// TIA Portal V19 program export: 1 tag tables, 0 data types, 0 data blocks, 3 code blocks (in call order from the OBs), 14 instance data blocks

VAR_GLOBAL   // PLC tag table "Default tag table"
   Axis_1_Drive_IN AT %I68.0 : "PD_TEL3_IN";
   Axis_1_Drive_OUT AT %Q82.0 : "PD_TEL3_OUT";
   "Axis_1_Homing switch" AT %I0.3 : Bool;
   firstscan AT %M10.0 : Bool;
   "Homing procedure" AT %M11.0 : Bool;
   Home_Done_Vertical AT %M11.1 : Bool;
   Tag_1 AT %I2.0 : Bool;
   Tag_2 AT %M20.0 : Bool;
   ServoONHorizont AT %Q0.7 : Bool;
   home_horizontal AT %Q0.4 : Bool;
   Home_done_horizontal AT %M12.0 : Bool;
   HomeComplete AT %I8.0 : Bool;
   Tag_3 AT %I1.3 : Bool;
   Servo_fault AT %I1.4 : Bool;
   Servo_Alarm AT %I1.5 : Bool;
   Tag_4 AT %M100.0 : Bool;
   System_Byte AT %MB8001 : Byte;
   "FirstScan(1)" AT %M1.0 : Bool;
   DiagStatusUpdate AT %M8001.1 : Bool;
   AlwaysTRUE AT %M8001.2 : Bool;
   AlwaysFALSE AT %M8001.3 : Bool;
   Clock_Byte AT %MB8000 : Byte;
   Clock_10Hz AT %M8000.0 : Bool;
   Clock_5Hz AT %M8000.1 : Bool;
   "Clock_2.5Hz" AT %M8000.2 : Bool;
   Clock_2Hz AT %M8000.3 : Bool;
   "Clock_1.25Hz" AT %M8000.4 : Bool;
   Clock_1Hz AT %M8000.5 : Bool;
   "Clock_0.625Hz" AT %M8000.6 : Bool;
   "Clock_0.5Hz" AT %M8000.7 : Bool;
   Tag_5 AT %M100.1 : Bool;
   Reset_HorizontDrive AT %Q0.6 : Bool;
   "hent 8cm" AT %M1000.0 : Bool;
   Binær_hent_8cm AT %M50.0 : Bool;
   Stepdata_1_U AT %Q0.1 : Bool;
   Stepdata_2_U AT %Q0.2 : Bool;
   Stepdata_3_U AT %Q0.3 : Bool;
   Stepdata_1_Conf AT %I0.6 : Bool;
   Stepdata_2_Conf AT %I0.7 : Bool;
   Stepdata_3_Conf AT %I1.0 : Bool;
   Drive_Servo AT %Q0.5 : Bool;
   lever_8cm AT %M1000.1 : Bool;
   "binær _lever_8cm" AT %M50.1 : Bool;
   "Sett sylinder C7" AT %M50.7 : Bool;
   "Sylinder C7" AT %Q0.0 : Bool;
   Tag_8 AT %M50.2 : Bool;
   Hent_16cm AT %M50.4 : Bool;
   Binær_Hent_16cm AT %M50.5 : Bool;
   Lever_16cm AT %M50.6 : Bool;
   binær_lever_16cm AT %M51.0 : Bool;
END_VAR

ORGANIZATION_BLOCK "Main"   // OB1, LAD, ProgramCycle
TITLE = "Main Program Sweep (Cycle)"
{ S7_Optimized_Access := 'TRUE' }
// stored: SetENOAutomatically false
   VAR_INPUT
      Initial_Call : Bool;   // Initial call of this OB
      Remanence : Bool;   // =True, if remanent data are available
   END_VAR
   VAR_TEMP   // added for the SCL form of the ladder/FBD networks
      _w1 : Bool;
   END_VAR
BEGIN

REGION Network 1: Homing Vertical
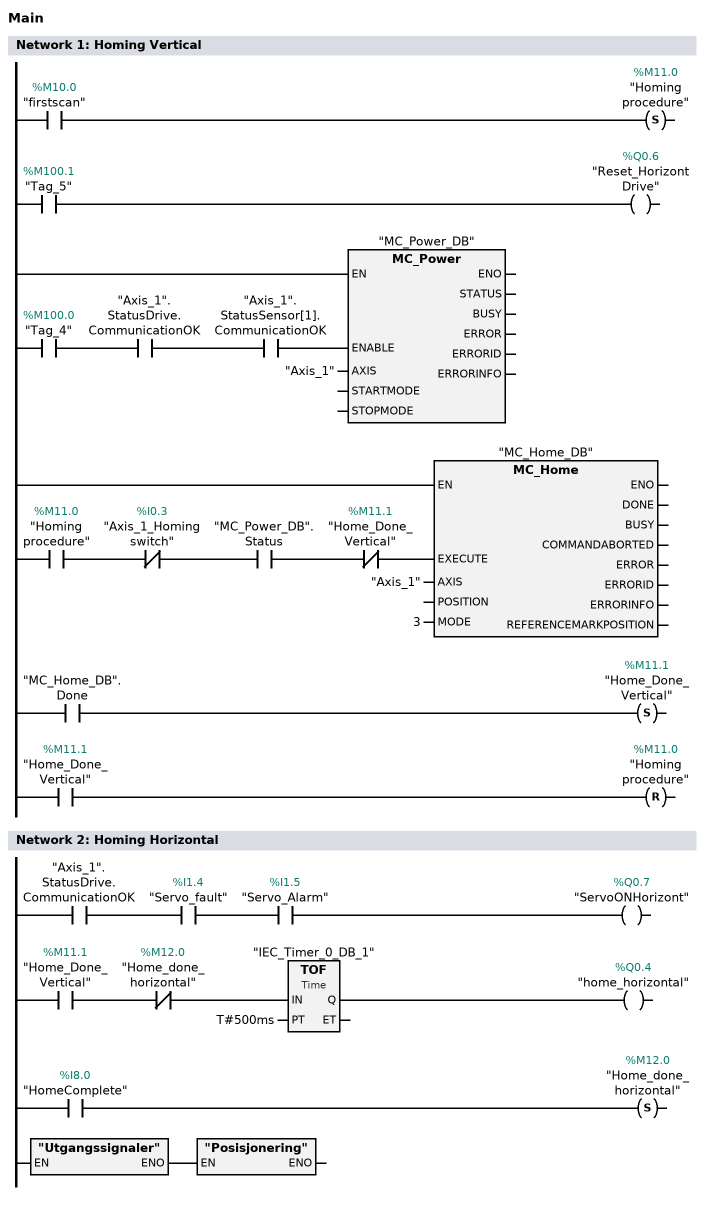
   RUNG wire#powerrail
      Contact( "firstscan" )
      S_Coil( "Homing procedure" )
   END_RUNG
   RUNG wire#powerrail
      Contact( "Tag_5" )
      Coil( "Reset_HorizontDrive" )
   END_RUNG
   RUNG wire#powerrail
      "MC_Power_DB".MC_Power(Enable := wire#w1, Axis := "Axis_1", StartMode :=, StopMode :=, Status =>, Busy =>, Error =>, ErrorID =>, ErrorInfo =>)
   END_RUNG
   RUNG wire#powerrail
      Contact( "Tag_4" )
      Contact( "Axis_1".StatusDrive.CommunicationOK )
      Contact( "Axis_1".StatusSensor[1].CommunicationOK )
   END_RUNG wire#w1
   RUNG wire#powerrail
      "MC_Home_DB".MC_Home(Execute := wire#w2, Axis := "Axis_1", Position :=, Mode := 3, Done =>, Busy =>, CommandAborted =>, Error =>, ErrorID =>, ErrorInfo =>, ReferenceMarkPosition =>)
   END_RUNG
   RUNG wire#powerrail
      Contact( "Homing procedure" )
      I_Contact( "Axis_1_Homing switch" )
      Contact( "MC_Power_DB".Status )
      I_Contact( "Home_Done_Vertical" )
   END_RUNG wire#w2
   RUNG wire#powerrail
      Contact( "MC_Home_DB".Done )
      S_Coil( "Home_Done_Vertical" )
   END_RUNG
   RUNG wire#powerrail
      Contact( "Home_Done_Vertical" )
      R_Coil( "Homing procedure" )
   END_RUNG
   // the same network as SCL:
   IF "firstscan" THEN "Homing procedure" := TRUE; END_IF;
   "Reset_HorizontDrive" := "Tag_5";
   "MC_Power_DB"(Enable := "Tag_4" AND "Axis_1".StatusDrive.CommunicationOK AND "Axis_1".StatusSensor[1].CommunicationOK,   // MC_Power
                 Axis := "Axis_1");
   "MC_Home_DB"(Execute := "Homing procedure" AND NOT "Axis_1_Homing switch" AND "MC_Power_DB".Status AND NOT "Home_Done_Vertical",   // MC_Home
                Axis := "Axis_1",
                Mode := 3);
   IF "MC_Home_DB".Done THEN "Home_Done_Vertical" := TRUE; END_IF;
   IF "Home_Done_Vertical" THEN "Homing procedure" := FALSE; END_IF;
END_REGION

REGION Network 2: Homing Horizontal
   RUNG wire#powerrail
      Contact( "Axis_1".StatusDrive.CommunicationOK )
      Contact( "Servo_fault" )
      Contact( "Servo_Alarm" )
      Coil( "ServoONHorizont" )
   END_RUNG
   RUNG wire#powerrail
      Contact( "Home_Done_Vertical" )
      I_Contact( "Home_done_horizontal" )
      { S7_Templates := "time_type := Time" } "IEC_Timer_0_DB_1".TOF(pt := T#500ms, et =>)
      Coil( "home_horizontal" )
   END_RUNG
   RUNG wire#powerrail
      Contact( "HomeComplete" )
      S_Coil( "Home_done_horizontal" )
   END_RUNG
   RUNG wire#powerrail
      "Utgangssignaler"()
      "Posisjonering"()
   END_RUNG
   // the same network as SCL:
   "ServoONHorizont" := "Axis_1".StatusDrive.CommunicationOK AND "Servo_fault" AND "Servo_Alarm";
   "IEC_Timer_0_DB_1".TOF(IN := "Home_Done_Vertical" AND NOT "Home_done_horizontal", PT := T#500ms);
   "home_horizontal" := "IEC_Timer_0_DB_1".Q;
   IF "HomeComplete" THEN "Home_done_horizontal" := TRUE; END_IF;
   "Utgangssignaler"(ENO => #_w1);
   IF #_w1 THEN "Posisjonering"(); END_IF;
END_REGION
END_ORGANIZATION_BLOCK

FUNCTION "Utgangssignaler" : Void   // FC1, LAD
{ S7_Optimized_Access := 'TRUE' }
// stored: SetENOAutomatically false
BEGIN

REGION Network 1
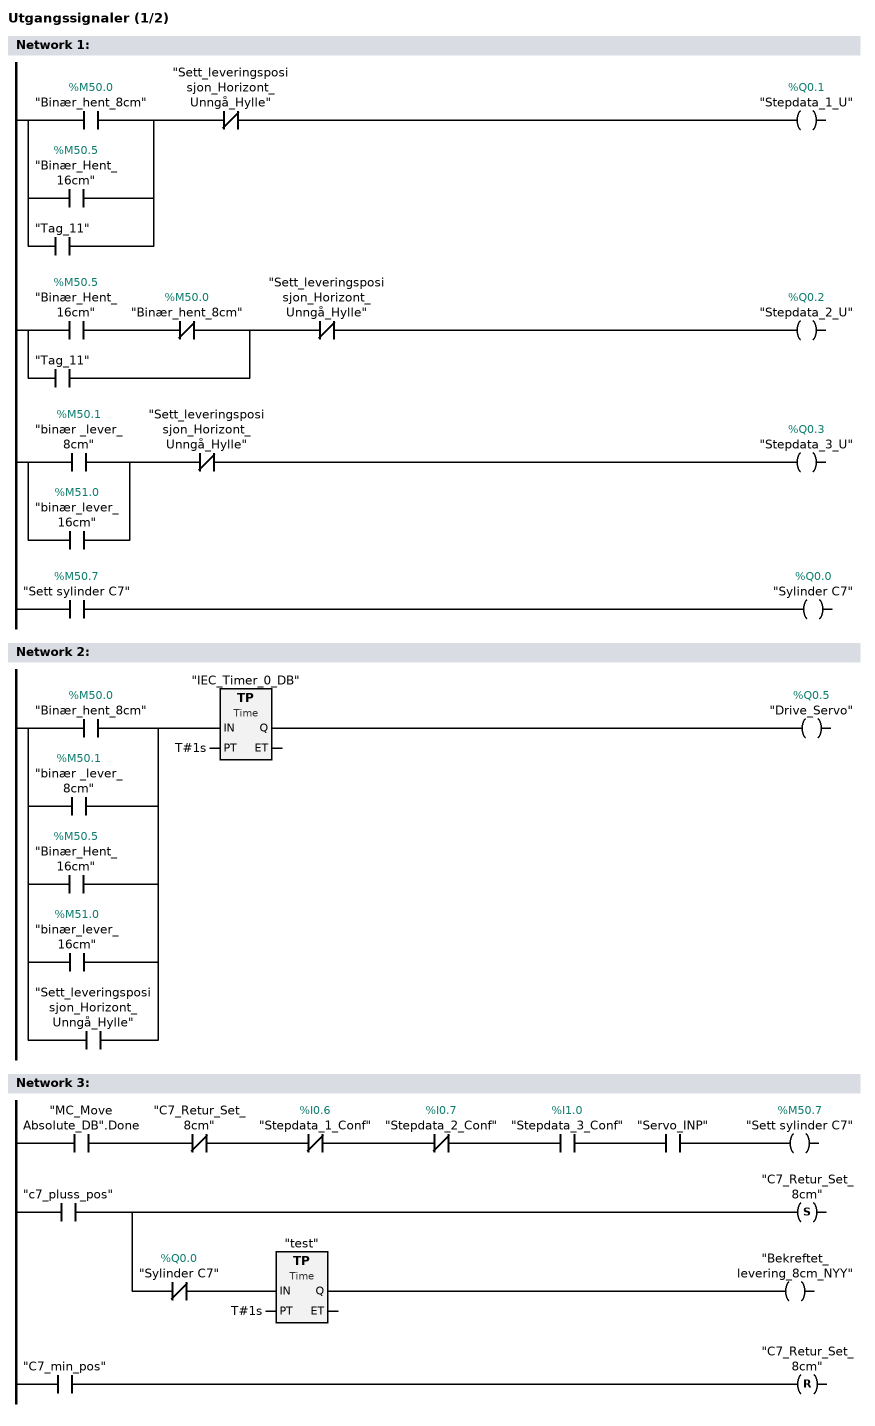
   RUNG wire#powerrail
      Contact( "Binær_hent_8cm" )
      wire#w1
      I_Contact( "Sett_leveringsposisjon_Horizont_Unngå_Hylle" )
      Coil( "Stepdata_1_U" )
   END_RUNG
   RUNG wire#powerrail
      Contact( "Binær_Hent_16cm" )
   END_RUNG wire#w1
   RUNG wire#powerrail
      Contact( "Tag_11" )
   END_RUNG wire#w1
   RUNG wire#powerrail
      Contact( "Binær_Hent_16cm" )
      I_Contact( "Binær_hent_8cm" )
      wire#w2
      I_Contact( "Sett_leveringsposisjon_Horizont_Unngå_Hylle" )
      Coil( "Stepdata_2_U" )
   END_RUNG
   RUNG wire#powerrail
      Contact( "Tag_11" )
   END_RUNG wire#w2
   RUNG wire#powerrail
      Contact( "binær _lever_8cm" )
      wire#w3
      I_Contact( "Sett_leveringsposisjon_Horizont_Unngå_Hylle" )
      Coil( "Stepdata_3_U" )
   END_RUNG
   RUNG wire#powerrail
      Contact( "binær_lever_16cm" )
   END_RUNG wire#w3
   RUNG wire#powerrail
      Contact( "Sett sylinder C7" )
      Coil( "Sylinder C7" )
   END_RUNG
   // the same network as SCL:
   "Stepdata_1_U" := ("Binær_hent_8cm" OR "Binær_Hent_16cm" OR "Tag_11") AND NOT "Sett_leveringsposisjon_Horizont_Unngå_Hylle";
   "Stepdata_2_U" := (("Binær_Hent_16cm" AND NOT "Binær_hent_8cm") OR "Tag_11") AND NOT "Sett_leveringsposisjon_Horizont_Unngå_Hylle";
   "Stepdata_3_U" := ("binær _lever_8cm" OR "binær_lever_16cm") AND NOT "Sett_leveringsposisjon_Horizont_Unngå_Hylle";
   "Sylinder C7" := "Sett sylinder C7";
END_REGION

REGION Network 2
   RUNG wire#powerrail
      Contact( "Binær_hent_8cm" )
      wire#w1
      { S7_Templates := "time_type := Time" } "IEC_Timer_0_DB".TP(pt := T#1s, et =>)
      Coil( "Drive_Servo" )
   END_RUNG
   RUNG wire#powerrail
      Contact( "binær _lever_8cm" )
   END_RUNG wire#w1
   RUNG wire#powerrail
      Contact( "Binær_Hent_16cm" )
   END_RUNG wire#w1
   RUNG wire#powerrail
      Contact( "binær_lever_16cm" )
   END_RUNG wire#w1
   RUNG wire#powerrail
      Contact( "Sett_leveringsposisjon_Horizont_Unngå_Hylle" )
   END_RUNG wire#w1
   // the same network as SCL:
   "IEC_Timer_0_DB".TP(IN := "Binær_hent_8cm" OR "binær _lever_8cm" OR "Binær_Hent_16cm" OR "binær_lever_16cm" OR "Sett_leveringsposisjon_Horizont_Unngå_Hylle",
                       PT := T#1s);
   "Drive_Servo" := "IEC_Timer_0_DB".Q;
END_REGION

REGION Network 3
   RUNG wire#powerrail
      Contact( "MC_MoveAbsolute_DB".Done )
      I_Contact( "C7_Retur_Set_8cm" )
      I_Contact( "Stepdata_1_Conf" )
      I_Contact( "Stepdata_2_Conf" )
      Contact( "Stepdata_3_Conf" )
      Contact( "Servo_INP" )
      Coil( "Sett sylinder C7" )
   END_RUNG
   RUNG wire#powerrail
      Contact( "c7_pluss_pos" )
      wire#w1
      S_Coil( "C7_Retur_Set_8cm" )
   END_RUNG
   RUNG wire#w1
      I_Contact( "Sylinder C7" )
      { S7_Templates := "time_type := Time" } "test".TP(pt := T#1s, et =>)
      Coil( "Bekreftet_levering_8cm_NYY" )
   END_RUNG
   RUNG wire#powerrail
      Contact( "C7_min_pos" )
      R_Coil( "C7_Retur_Set_8cm" )
   END_RUNG
   // the same network as SCL:
   "Sett sylinder C7" := "MC_MoveAbsolute_DB".Done AND NOT "C7_Retur_Set_8cm" AND NOT "Stepdata_1_Conf" AND NOT "Stepdata_2_Conf" AND "Stepdata_3_Conf" AND "Servo_INP";
   IF "c7_pluss_pos" THEN "C7_Retur_Set_8cm" := TRUE; END_IF;
   "test".TP(IN := "c7_pluss_pos" AND NOT "Sylinder C7", PT := T#1s);
   "Bekreftet_levering_8cm_NYY" := "test".Q;
   IF "C7_min_pos" THEN "C7_Retur_Set_8cm" := FALSE; END_IF;
END_REGION

REGION Network 4
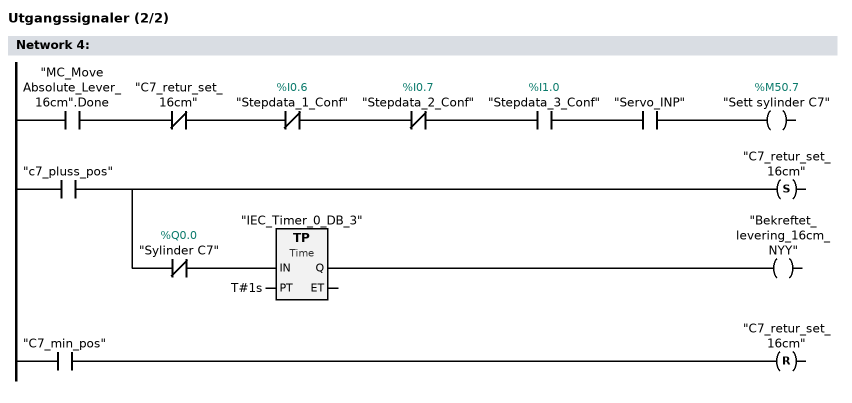
   RUNG wire#powerrail
      Contact( "MC_MoveAbsolute_Lever_16cm".Done )
      I_Contact( "C7_retur_set_16cm" )
      I_Contact( "Stepdata_1_Conf" )
      I_Contact( "Stepdata_2_Conf" )
      Contact( "Stepdata_3_Conf" )
      Contact( "Servo_INP" )
      Coil( "Sett sylinder C7" )
   END_RUNG
   RUNG wire#powerrail
      Contact( "c7_pluss_pos" )
      wire#w1
      S_Coil( "C7_retur_set_16cm" )
   END_RUNG
   RUNG wire#w1
      I_Contact( "Sylinder C7" )
      { S7_Templates := "time_type := Time" } "IEC_Timer_0_DB_3".TP(pt := T#1s, et =>)
      Coil( "Bekreftet_levering_16cm_NYY" )
   END_RUNG
   RUNG wire#powerrail
      Contact( "C7_min_pos" )
      R_Coil( "C7_retur_set_16cm" )
   END_RUNG
   // the same network as SCL:
   "Sett sylinder C7" := "MC_MoveAbsolute_Lever_16cm".Done AND NOT "C7_retur_set_16cm" AND NOT "Stepdata_1_Conf" AND NOT "Stepdata_2_Conf" AND "Stepdata_3_Conf" AND "Servo_INP";
   IF "c7_pluss_pos" THEN "C7_retur_set_16cm" := TRUE; END_IF;
   "IEC_Timer_0_DB_3".TP(IN := "c7_pluss_pos" AND NOT "Sylinder C7", PT := T#1s);
   "Bekreftet_levering_16cm_NYY" := "IEC_Timer_0_DB_3".Q;
   IF "C7_min_pos" THEN "C7_retur_set_16cm" := FALSE; END_IF;
END_REGION
END_FUNCTION

FUNCTION "Posisjonering" : Void   // FC2, LAD
{ S7_Optimized_Access := 'TRUE' }
// stored: SetENOAutomatically false
BEGIN

REGION Network 1
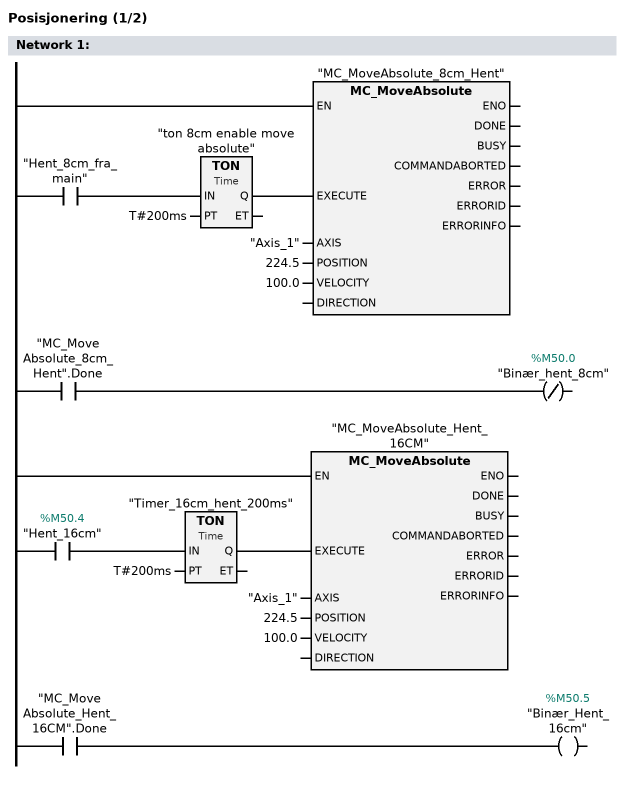
   RUNG wire#powerrail
      "MC_MoveAbsolute_8cm_Hent".MC_MoveAbsolute(Execute := wire#w1, Axis := "Axis_1", Position := 224.5, Velocity := 100.0, Direction :=, Done =>, Busy =>, CommandAborted =>, Error =>, ErrorID =>, ErrorInfo =>)
   END_RUNG
   RUNG wire#powerrail
      Contact( "Hent_8cm_fra_main" )
      { S7_Templates := "time_type := Time" } "ton 8cm enable move absolute".TON(pt := T#200ms, et =>)
   END_RUNG wire#w1
   RUNG wire#powerrail
      Contact( "MC_MoveAbsolute_8cm_Hent".Done )
      I_Coil( "Binær_hent_8cm" )
   END_RUNG
   RUNG wire#powerrail
      "MC_MoveAbsolute_Hent_16CM".MC_MoveAbsolute(Execute := wire#w2, Axis := "Axis_1", Position := 224.5, Velocity := 100.0, Direction :=, Done =>, Busy =>, CommandAborted =>, Error =>, ErrorID =>, ErrorInfo =>)
   END_RUNG
   RUNG wire#powerrail
      Contact( "Hent_16cm" )
      { S7_Templates := "time_type := Time" } "Timer_16cm_hent_200ms".TON(pt := T#200ms, et =>)
   END_RUNG wire#w2
   RUNG wire#powerrail
      Contact( "MC_MoveAbsolute_Hent_16CM".Done )
      Coil( "Binær_Hent_16cm" )
   END_RUNG
   // the same network as SCL:
   "ton 8cm enable move absolute".TON(IN := "Hent_8cm_fra_main", PT := T#200ms);
   "MC_MoveAbsolute_8cm_Hent"(Execute := "ton 8cm enable move absolute".Q,   // MC_MoveAbsolute
                           Axis := "Axis_1",
                           Position := 224.5,
                           Velocity := 100.0);
   "Binær_hent_8cm" := NOT "MC_MoveAbsolute_8cm_Hent".Done;
   "Timer_16cm_hent_200ms".TON(IN := "Hent_16cm", PT := T#200ms);
   "MC_MoveAbsolute_Hent_16CM"(Execute := "Timer_16cm_hent_200ms".Q,   // MC_MoveAbsolute
                           Axis := "Axis_1",
                           Position := 224.5,
                           Velocity := 100.0);
   "Binær_Hent_16cm" := "MC_MoveAbsolute_Hent_16CM".Done;
END_REGION

REGION Network 2
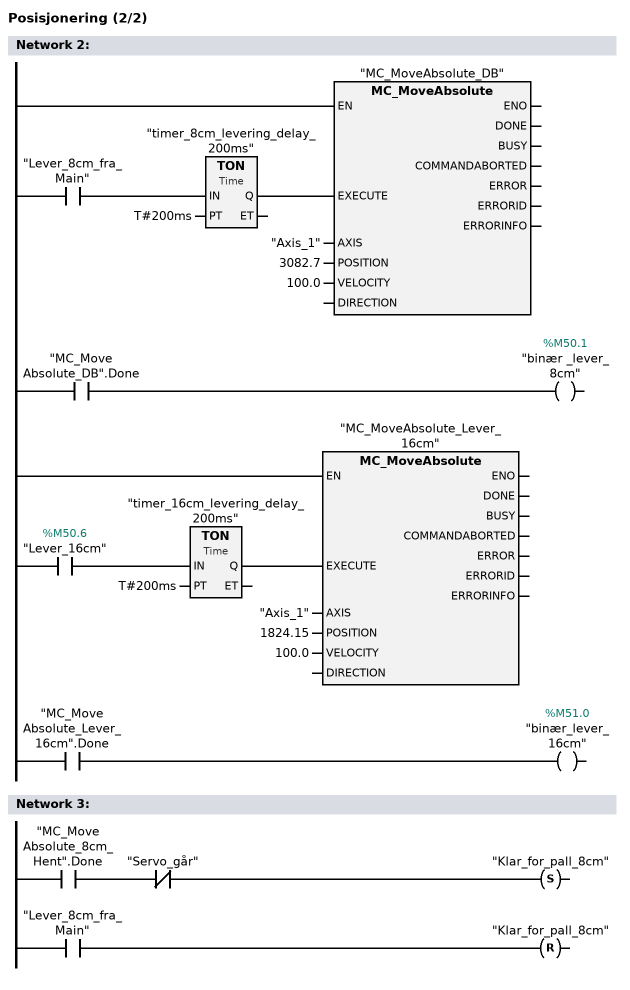
   RUNG wire#powerrail
      "MC_MoveAbsolute_DB".MC_MoveAbsolute(Execute := wire#w1, Axis := "Axis_1", Position := 3082.7, Velocity := 100.0, Direction :=, Done =>, Busy =>, CommandAborted =>, Error =>, ErrorID =>, ErrorInfo =>)
   END_RUNG
   RUNG wire#powerrail
      Contact( "Lever_8cm_fra_Main" )
      { S7_Templates := "time_type := Time" } "timer_8cm_levering_delay_200ms".TON(pt := T#200ms, et =>)
   END_RUNG wire#w1
   RUNG wire#powerrail
      Contact( "MC_MoveAbsolute_DB".Done )
      Coil( "binær _lever_8cm" )
   END_RUNG
   RUNG wire#powerrail
      "MC_MoveAbsolute_Lever_16cm".MC_MoveAbsolute(Execute := wire#w2, Axis := "Axis_1", Position := 1824.15, Velocity := 100.0, Direction :=, Done =>, Busy =>, CommandAborted =>, Error =>, ErrorID =>, ErrorInfo =>)
   END_RUNG
   RUNG wire#powerrail
      Contact( "Lever_16cm" )
      { S7_Templates := "time_type := Time" } "timer_16cm_levering_delay_200ms".TON(pt := T#200ms, et =>)
   END_RUNG wire#w2
   RUNG wire#powerrail
      Contact( "MC_MoveAbsolute_Lever_16cm".Done )
      Coil( "binær_lever_16cm" )
   END_RUNG
   // the same network as SCL:
   "timer_8cm_levering_delay_200ms".TON(IN := "Lever_8cm_fra_Main", PT := T#200ms);
   "MC_MoveAbsolute_DB"(Execute := "timer_8cm_levering_delay_200ms".Q,   // MC_MoveAbsolute
                        Axis := "Axis_1",
                        Position := 3082.7,
                        Velocity := 100.0);
   "binær _lever_8cm" := "MC_MoveAbsolute_DB".Done;
   "timer_16cm_levering_delay_200ms".TON(IN := "Lever_16cm", PT := T#200ms);
   "MC_MoveAbsolute_Lever_16cm"(Execute := "timer_16cm_levering_delay_200ms".Q,   // MC_MoveAbsolute
                           Axis := "Axis_1",
                           Position := 1824.15,
                           Velocity := 100.0);
   "binær_lever_16cm" := "MC_MoveAbsolute_Lever_16cm".Done;
END_REGION

REGION Network 3
   RUNG wire#powerrail
      Contact( "MC_MoveAbsolute_8cm_Hent".Done )
      I_Contact( "Servo_går" )
      S_Coil( "Klar_for_pall_8cm" )
   END_RUNG
   RUNG wire#powerrail
      Contact( "Lever_8cm_fra_Main" )
      R_Coil( "Klar_for_pall_8cm" )
   END_RUNG
   // the same network as SCL:
   IF "MC_MoveAbsolute_8cm_Hent".Done AND NOT "Servo_går" THEN "Klar_for_pall_8cm" := TRUE; END_IF;
   IF "Lever_8cm_fra_Main" THEN "Klar_for_pall_8cm" := FALSE; END_IF;
END_REGION
END_FUNCTION

DATA_BLOCK "Home delay firstscan"   // DB8
{ S7_Optimized_Access := 'TRUE' }
// stored: InstanceOfName IEC_TIMER, OfSystemLibElement IEC_TIMER, OfSystemLibVersion 1.0
"IEC_TIMER"
   // VAR
   //    PT : Time;
   //    ET { ExternalWritable := 'False'} : Time;
   //    IN : Bool;
   //    Q { ExternalWritable := 'False'} : Bool;
   // END_VAR
BEGIN
END_DATA_BLOCK

DATA_BLOCK "IEC_Timer_0_DB"   // DB4
{ S7_Optimized_Access := 'TRUE' }
// stored: InstanceOfName IEC_TIMER, OfSystemLibElement IEC_TIMER, OfSystemLibVersion 1.0
"IEC_TIMER"
   // VAR
   //    PT : Time;
   //    ET { ExternalWritable := 'False'} : Time;
   //    IN : Bool;
   //    Q { ExternalWritable := 'False'} : Bool;
   // END_VAR
BEGIN
END_DATA_BLOCK

DATA_BLOCK "IEC_Timer_0_DB_1"   // DB6
{ S7_Optimized_Access := 'TRUE' }
// stored: InstanceOfName IEC_TIMER, OfSystemLibElement IEC_TIMER, OfSystemLibVersion 1.0
"IEC_TIMER"
   // VAR
   //    PT : Time;
   //    ET { ExternalWritable := 'False'} : Time;
   //    IN : Bool;
   //    Q { ExternalWritable := 'False'} : Bool;
   // END_VAR
BEGIN
END_DATA_BLOCK

DATA_BLOCK "MC_Home_DB"   // DB3
// stored: InstanceOfName MC_Home, OfSystemLibElement MC_Home, OfSystemLibVersion 7.0
"MC_Home"
   // VAR_INPUT
   //    Axis : TO_Axis;
   //    Execute : Bool;
   //    Position : Real;
   //    Mode : Int;
   // END_VAR
   // VAR_OUTPUT
   //    Done : Bool;
   //    Busy : Bool;
   //    CommandAborted : Bool;
   //    Error : Bool;
   //    ErrorID : Word;
   //    ErrorInfo : Word;
   //    ReferenceMarkPosition : Real;
   // END_VAR
   // VAR
   //    FB_ID : DInt;
   // END_VAR
BEGIN
END_DATA_BLOCK

DATA_BLOCK "MC_MoveAbsolute_8cm_Hent"   // DB7
// stored: InstanceOfName MC_MoveAbsolute, OfSystemLibElement MC_MoveAbsolute, OfSystemLibVersion 7.0
"MC_MoveAbsolute"
   // VAR_INPUT
   //    Axis : TO_PositioningAxis;
   //    Execute : Bool;
   //    Position : Real;
   //    Velocity : Real;
   //    Direction : Int;
   // END_VAR
   // VAR_OUTPUT
   //    Done : Bool;
   //    Busy : Bool;
   //    CommandAborted : Bool;
   //    Error : Bool;
   //    ErrorID : Word;
   //    ErrorInfo : Word;
   // END_VAR
   // VAR
   //    FB_ID : DInt;
   // END_VAR
BEGIN
END_DATA_BLOCK

DATA_BLOCK "MC_MoveAbsolute_DB"   // DB9
// stored: InstanceOfName MC_MoveAbsolute, OfSystemLibElement MC_MoveAbsolute, OfSystemLibVersion 7.0
"MC_MoveAbsolute"
   // VAR_INPUT
   //    Axis : TO_PositioningAxis;
   //    Execute : Bool;
   //    Position : Real;
   //    Velocity : Real;
   //    Direction : Int;
   // END_VAR
   // VAR_OUTPUT
   //    Done : Bool;
   //    Busy : Bool;
   //    CommandAborted : Bool;
   //    Error : Bool;
   //    ErrorID : Word;
   //    ErrorInfo : Word;
   // END_VAR
   // VAR
   //    FB_ID : DInt;
   // END_VAR
BEGIN
END_DATA_BLOCK

DATA_BLOCK "MC_MoveAbsolute_Hent_16CM"   // DB11
// stored: InstanceOfName MC_MoveAbsolute, OfSystemLibElement MC_MoveAbsolute, OfSystemLibVersion 7.0
"MC_MoveAbsolute"
   // VAR_INPUT
   //    Axis : TO_PositioningAxis;
   //    Execute : Bool;
   //    Position : Real;
   //    Velocity : Real;
   //    Direction : Int;
   // END_VAR
   // VAR_OUTPUT
   //    Done : Bool;
   //    Busy : Bool;
   //    CommandAborted : Bool;
   //    Error : Bool;
   //    ErrorID : Word;
   //    ErrorInfo : Word;
   // END_VAR
   // VAR
   //    FB_ID : DInt;
   // END_VAR
BEGIN
END_DATA_BLOCK

DATA_BLOCK "MC_MoveAbsolute_Lever_16cm"   // DB13
// stored: InstanceOfName MC_MoveAbsolute, OfSystemLibElement MC_MoveAbsolute, OfSystemLibVersion 7.0
"MC_MoveAbsolute"
   // VAR_INPUT
   //    Axis : TO_PositioningAxis;
   //    Execute : Bool;
   //    Position : Real;
   //    Velocity : Real;
   //    Direction : Int;
   // END_VAR
   // VAR_OUTPUT
   //    Done : Bool;
   //    Busy : Bool;
   //    CommandAborted : Bool;
   //    Error : Bool;
   //    ErrorID : Word;
   //    ErrorInfo : Word;
   // END_VAR
   // VAR
   //    FB_ID : DInt;
   // END_VAR
BEGIN
END_DATA_BLOCK

DATA_BLOCK "MC_Power_DB"   // DB2
// stored: InstanceOfName MC_Power, OfSystemLibElement MC_Power, OfSystemLibVersion 7.0
"MC_Power"
   // VAR_INPUT
   //    Axis : TO_Axis;
   //    Enable : Bool;
   //    StartMode : Int;
   //    StopMode : Int;
   // END_VAR
   // VAR_OUTPUT
   //    Status : Bool;
   //    Busy : Bool;
   //    Error : Bool;
   //    ErrorID : Word;
   //    ErrorInfo : Word;
   // END_VAR
   // VAR
   //    FB_ID : DInt;
   // END_VAR
BEGIN
END_DATA_BLOCK

DATA_BLOCK "Timer_16cm_hent_200ms"   // DB12
{ S7_Optimized_Access := 'TRUE' }
// stored: InstanceOfName IEC_TIMER, OfSystemLibElement IEC_TIMER, OfSystemLibVersion 1.0
"IEC_TIMER"
   // VAR
   //    PT : Time;
   //    ET { ExternalWritable := 'False'} : Time;
   //    IN : Bool;
   //    Q { ExternalWritable := 'False'} : Bool;
   // END_VAR
BEGIN
END_DATA_BLOCK

DATA_BLOCK "timer_16cm_levering_delay_200ms"   // DB14
{ S7_Optimized_Access := 'TRUE' }
// stored: InstanceOfName IEC_TIMER, OfSystemLibElement IEC_TIMER, OfSystemLibVersion 1.0
"IEC_TIMER"
   // VAR
   //    PT : Time;
   //    ET { ExternalWritable := 'False'} : Time;
   //    IN : Bool;
   //    Q { ExternalWritable := 'False'} : Bool;
   // END_VAR
BEGIN
END_DATA_BLOCK

DATA_BLOCK "timer_8cm_levering_delay_200ms"   // DB10
{ S7_Optimized_Access := 'TRUE' }
// stored: InstanceOfName IEC_TIMER, OfSystemLibElement IEC_TIMER, OfSystemLibVersion 1.0
"IEC_TIMER"
   // VAR
   //    PT : Time;
   //    ET { ExternalWritable := 'False'} : Time;
   //    IN : Bool;
   //    Q { ExternalWritable := 'False'} : Bool;
   // END_VAR
BEGIN
END_DATA_BLOCK

DATA_BLOCK "ton 8cm enable move absolute"   // DB5
{ S7_Optimized_Access := 'TRUE' }
// stored: InstanceOfName IEC_TIMER, OfSystemLibElement IEC_TIMER, OfSystemLibVersion 1.0
"IEC_TIMER"
   // VAR
   //    PT : Time;
   //    ET { ExternalWritable := 'False'} : Time;
   //    IN : Bool;
   //    Q { ExternalWritable := 'False'} : Bool;
   // END_VAR
BEGIN
END_DATA_BLOCK

DATA_BLOCK "Axis_1"   // DB1, Motion_DB
AUTHOR : SIMATIC
FAMILY : BasicMC
NAME : TO_PosAx
VERSION : 7.0
// stored: InstanceOfName TO_PositioningAxis, OfSystemLibElement TO_PositioningAxis, OfSystemLibVersion 7.0
TO_PositioningAxis   // technology object, version 7.0
   // // inherited from TO_SpeedAxis
   // // inherited from TO_Axis
   // // inherited from TO_AnyMotionObject
   // VAR
   //    Header : TO_Struct_Header;
   // END_VAR
   // VAR
   //    Position { ExternalWritable := 'False'} : Real;
   //    Velocity { ExternalWritable := 'False'} : Real;
   //    ActualPosition { ExternalWritable := 'False'} : Real;
   //    ActualVelocity { ExternalWritable := 'False'} : Real;
   //    Actor { S7_SetPoint := 'True'} : TO_Struct_Actor;
   //    Sensor { S7_SetPoint := 'True'} : Array[1..1] of TO_Struct_Sensor;
   //    Units { ExternalWritable := 'False'; S7_SetPoint := 'True'} : TO_Struct_Units;
   //    Mechanics { ExternalWritable := 'False'; S7_SetPoint := 'True'} : TO_Struct_Mechanics;
   //    DynamicLimits { ExternalWritable := 'False'; S7_SetPoint := 'True'} : TO_Struct_DynamicLimits;
   //    DynamicDefaults { S7_SetPoint := 'True'} : TO_Struct_DynamicDefaults;
   //    Modulo { ExternalWritable := 'False'; S7_SetPoint := 'True'} : TO_Struct_Modulo;
   //    PositionLimits_SW { S7_SetPoint := 'True'} : TO_Struct_PositionLimitsSW;
   //    PositionLimits_HW { S7_SetPoint := 'True'} : TO_Struct_PositionLimitsHW;
   //    Homing { S7_SetPoint := 'True'} : TO_Struct_Homing;
   //    PositionControl { ExternalWritable := 'False'; S7_SetPoint := 'True'} : TO_Struct_PositionControl;
   //    FollowingError { ExternalWritable := 'False'; S7_SetPoint := 'True'} : TO_Struct_FollowingError;
   //    PositioningMonitoring { ExternalWritable := 'False'; S7_SetPoint := 'True'} : TO_Struct_PositioningMonitoring;
   //    StandstillSignal { ExternalWritable := 'False'; S7_SetPoint := 'True'} : TO_Struct_StandstillSignal;
   //    Simulation { ExternalWritable := 'False'; S7_SetPoint := 'True'} : TO_Struct_Simulation;
   //    StatusPositioning { ExternalWritable := 'False'; S7_SetPoint := 'True'} : TO_Struct_StatusPositioning;
   //    StatusDrive { ExternalWritable := 'False'; S7_SetPoint := 'True'} : TO_Struct_StatusDrive;
   //    StatusSensor { ExternalWritable := 'False'; S7_SetPoint := 'True'} : Array[1..1] of TO_Struct_StatusSensor;
   //    StatusBits { ExternalWritable := 'False'; S7_SetPoint := 'True'} : TO_Struct_StatusBits;
   //    ErrorBits { ExternalWritable := 'False'; S7_SetPoint := 'True'} : TO_Struct_ErrorBits;
   //    ControlPanel { S7_SetPoint := 'True'} : TO_Struct_ControlPanel;
   //    Internal { S7_SetPoint := 'True'} : Array[1..4] of TO_Struct_Internal;
   // END_VAR
BEGIN
   Header.VersionMaj := 7;
   Header.VersionMin := 0;
   Header."Type" := 1;
   Actor."Type" := 1;
   Actor.DataAdaption := 1;
   Actor.Interface.AddressIn.RID := 16#0208_070C;
   Actor.Interface.AddressIn.AREA := 16#81;
   Actor.Interface.AddressIn.OFFSET := 544;
   Actor.Interface.AddressOut.RID := 16#0208_070D;
   Actor.Interface.AddressOut.AREA := 16#82;
   Actor.Interface.AddressOut.OFFSET := 656;
   Actor.DriveParameter.MaxSpeed := 5000.0;
   Sensor[1].DataAdaption := 1;
   Sensor[1].Interface.AddressIn.RID := 16#0208_070C;
   Sensor[1].Interface.AddressIn.AREA := 16#81;
   Sensor[1].Interface.AddressIn.OFFSET := 544;
   Sensor[1].Interface.AddressOut.RID := 16#0208_070D;
   Sensor[1].Interface.AddressOut.AREA := 16#82;
   Sensor[1].Interface.AddressOut.OFFSET := 656;
   Sensor[1].Interface."Type" := 2;
   Sensor[1].Parameter.StepsPerRevolution := 2500;
   Sensor[1].Parameter.FineResolutionXist1 := 2;
   Sensor[1].Parameter.FineResolutionXist2 := 0;
   Sensor[1].Parameter.DeterminableRevolutions := 0;
   Sensor[1].ActiveHoming.DigitalInputAddress.RID := 16#0200_0001;
   Sensor[1].ActiveHoming.DigitalInputAddress.AREA := 16#81;
   Sensor[1].ActiveHoming.DigitalInputAddress.OFFSET := 3;
   Sensor[1].ActiveHoming.SwitchLevel := FALSE;
   DynamicLimits.MinVelocity := 0.0;
   DynamicDefaults.Acceleration := 50.0;
   DynamicDefaults.Deceleration := 50.0;
   DynamicDefaults.EmergencyDeceleration := 125.0;
   Homing.AutoReversal := FALSE;
   Homing.ApproachDirection := FALSE;
   _Sensor[1].ActiveHoming.DigitalInput := Axis_1_Homing switch;
   _Sensor[1].DataAdaptionOffline := True;
   _Sensor[1].Interface.ProfiDriveOutName := Axis_1_Drive_OUT;
   _Sensor[1].Interface.ProfiDriveInName := Axis_1_Drive_IN;
   _Actor.DataAdaptionOffline := True;
   _Actor.Interface.ProfiDriveOutName := Axis_1_Drive_OUT;
   _Actor.Interface.ProfiDriveInName := Axis_1_Drive_IN;
   _Sensor[1].Interface.EncoderConnection := 7;
END_DATA_BLOCK
